// SIMATIC S7-200 project (STEP 7-Micro/WIN), CPU 226 REL 02.01

SYMBOL_TABLE 用户定义1
步进启动             I0.0
步进停止             I0.1
脉冲输出             Q0.0
步进循环             T37
总脉冲数             SMD72
定义周期             SMW68
定义控制             SMB67
脉冲结束             SM66.7
END_SYMBOL_TABLE

ORGANIZATION_BLOCK 主程序:OB1
TITLE=程序注释
BEGIN
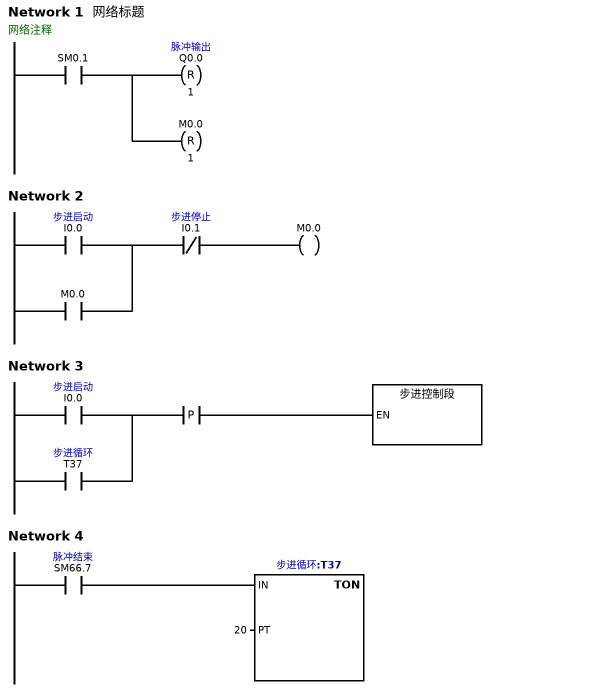
Network 1 // 网络标题
// 网络注释
LD     SM0.1
R      脉冲输出:Q0.0, 1
R      M0.0, 1
Network 2
LD     步进启动:I0.0
O      M0.0
AN     步进停止:I0.1
=      M0.0
Network 3
LD     步进启动:I0.0
O      步进循环:T37
EU
CALL   步进控制段:SBR0
Network 4
LD     脉冲结束:SM66.7
TON    步进循环:T37, 20
END_ORGANIZATION_BLOCK

SUBROUTINE_BLOCK 步进控制段:SBR0
TITLE=子程序注释
BEGIN
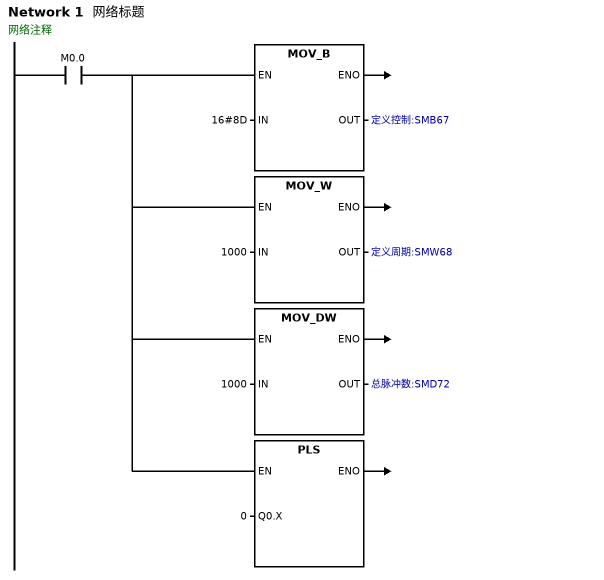
Network 1 // 网络标题
// 网络注释
LD     M0.0
MOVB   16#8D, 定义控制:SMB67
MOVW   1000, 定义周期:SMW68
MOVD   1000, 总脉冲数:SMD72
PLS    0
END_SUBROUTINE_BLOCK
